// TIA Portal V20 export
ORGANIZATION_BLOCK "Main"   // OB1011, LAD, ProgramCycle
TITLE = "Main Program Sweep (Cycle)"
AUTHOR : ERsystem_FA2_DH. Kim
// stored: AutoNumber false, IsIECCheckEnabled true, Namespace Unit1.Em1, SetENOAutomatically false
   VAR_INPUT
      Initial_Call : Bool;   // Initial call of this OB
      Remanence : Bool;   // =True, if remanent data are available
   END_VAR
   VAR_TEMP
      tempIndex : Int;   // Index of EM in the array
   END_VAR
BEGIN

REGION Network 1
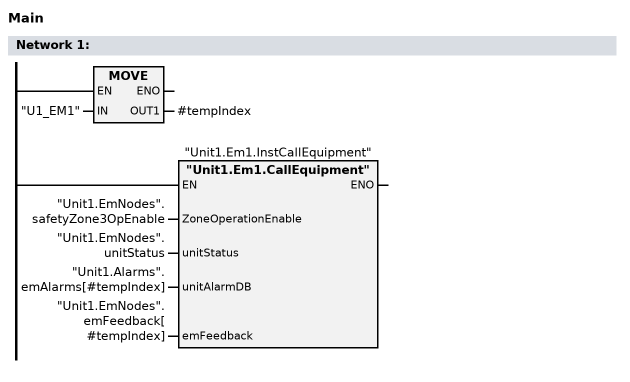
   RUNG wire#powerrail
      Move(in := "U1_EM1", out1 => #tempIndex)
   END_RUNG
   RUNG wire#powerrail
      "Unit1.Em1.InstCallEquipment"(ZoneOperationEnable := "Unit1.EmNodes".safetyZone3OpEnable, unitStatus := "Unit1.EmNodes".unitStatus, unitAlarmDB := "Unit1.Alarms".emAlarms[#tempIndex], emFeedback := "Unit1.EmNodes".emFeedback[#tempIndex])
   END_RUNG
   // the same network as SCL:
   #tempIndex := "U1_EM1";
   "Unit1.Em1.InstCallEquipment"(ZoneOperationEnable := "Unit1.EmNodes".safetyZone3OpEnable,   // "Unit1.Em1.CallEquipment"
                           unitStatus := "Unit1.EmNodes".unitStatus,
                           unitAlarmDB := "Unit1.Alarms".emAlarms[#tempIndex],
                           emFeedback := "Unit1.EmNodes".emFeedback[#tempIndex]);
END_REGION
END_ORGANIZATION_BLOCK
